// TIA Portal V20 export
TYPE "IO_VLV"
   STRUCT
      IN { ExternalAccessible := 'False'; ExternalVisible := 'False'; ExternalWritable := 'False'} : Struct
         OpenFb : Bool;
         ClosedFb : Bool;
         Fault : Bool;
      END_STRUCT;
      OUT { ExternalAccessible := 'False'; ExternalVisible := 'False'; ExternalWritable := 'False'} : Struct
         OpenCmd : Bool;
         CloseCmd : Bool;
      END_STRUCT;
   END_STRUCT;
END_TYPE
